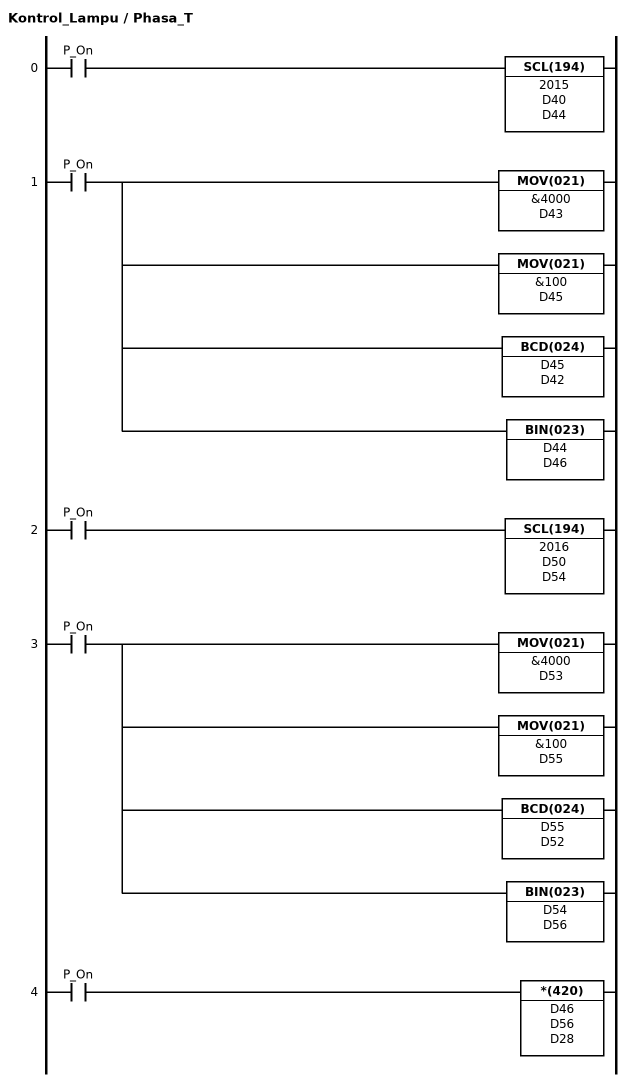
; [picture p24: Kontrol_Lampu / Phasa_T, rungs 0-4]
; rung 0
LD P_On
SCL(194) 2015 D40 D44
; rung 1
LD P_On
MOV(021) &4000 D43
MOV(021) &100 D45
BCD(024) D45 D42
BIN(023) D44 D46
; rung 2
LD P_On
SCL(194) 2016 D50 D54
; rung 3
LD P_On
MOV(021) &4000 D53
MOV(021) &100 D55
BCD(024) D55 D52
BIN(023) D54 D56
; rung 4
LD P_On
*(420) D46 D56 D28

### Section END
; rung 0
END(001)